FUNCTION F_ITC_SendIPR : BOOL
(**************************************************************************************
 * 	Application		:	BoxControl Framework
 *	Revision		:	$Revision: 404529 $
 *	Revision date	:	$Date: 2018-04-23 08:21:38 +0200 (Mo., 23 Apr 2018) $
 *	Last changed by	:	$Author: b7bolm $
 *	URL				:	$URL: http://almscdc.swisslog.com/repo/SWPD/Development/BoxControlFramework/20_Release/trunk/01_Software/BCF/BCF/JumpStart/20_Product/10_App/11_Com/10_Lib/10_Conv/11_ITC/F_ITC_SendIPR.TcPOU $
 *
 *	Purpose			:	Wrap message - IPR
 *
 * ------------------------------------------------------------------------------------
 *	Copyright Swisslog [IP AG], Switzerland. All rights reserved.
 * 
 * ------------------------------------------------------------------------------------
 *	
 * 	Revision History: 
 *
 * 	VERSION			DATE			INITIALS			DESCRIPTION
 *	0.1				01.01.2001		swl					Example
 *
 **************************************************************************************)
VAR_INPUT
	eChannelSrc			: E_MFCS_Channel; // Source communicaton channel
	Position			: STRING(Conveyor.POSITION_STRINGLENGTH); // SIS MM-GGG-EEEE-FF-Z
	TU_DataIndex		: DINT; // TU-DataIndex
	MSG_Sequence		: INT; // Assignment message sequence
	TU_ID				: STRING(Conveyor.TU_ID_STRINGLENGTH); // 18 Char SSID
	TU_Type				: INT; // TU-Type
	AssignmentID		: UDINT; // Assignment id
	Height				: INT; // Height Result
	WidthRight			: INT; // Width Right Result
	WidthLeft			: INT; // Width Left Result
	LengthFront			: INT; // Length Front Result
	LengthRear			: INT; // Length Rear Result
	Weight				: DINT; // Weight Value
	Tunnel				: INT; // Tunnel Result
	Runner				: INT; // Runner Result
	ErrorCode			: INT; // Error
	ValidLabelString	: INT; // Valid Label Return Code
	Label				: STRING(Conveyor.LABEL_LENGTH); // Characters of Label Data
END_VAR
VAR
	IPR					: ST_ITC_IPR; 
END_VAR

// Map values
IPR.Position := Position;
IPR.TU_DataIndex := TU_DataIndex;
IPR.MSG_Sequence := MSG_Sequence;
IPR.TU_ID := TU_ID;
IPR.TU_Type := TU_Type;
IPR.AssignmentID := AssignmentID;
IPR.Height := Height;
IPR.WidthRight := WidthRight;
IPR.WidthLeft := WidthLeft;
IPR.LengthFront := LengthFront;
IPR.LengthRear := LengthRear;
IPR.Weight := Weight;
IPR.Tunnel := Tunnel;
IPR.Runner := Runner;
IPR.ErrorCode := ErrorCode;
IPR.ValidLabelString := ValidLabelString;
IPR.Label := Label;

// Forward to ITC
F_ITC_SendIPR := fbITC_Manager.M_SendData(
					meChannel	:= eChannelSrc,
					mMsgType	:= E_ITC_MsgTypeConv.IDENTIFICATION_REPORT,
					mpData		:= ADR(IPR),
					mLen		:= SIZEOF(IPR));

END_FUNCTION

(* stored: Version 1.1.0.1, ProductVersion 3.1.4022.12
   POU F_ITC_SendIPR: Id {4cd04075-63d3-4a01-a5b4-9f44deb85d64}, SpecialFunc None *)
